Fanuc KAREL source: kc00049.KL

-- PROVISIONAL review KL for V1013-1; original PC SHA256 6f2dececdb086ac4d14ee3edc9f621b24aaa7305749a3dd8db25e0824419496a
-- Incomplete behavior may be omitted. Consult companion uncertainty JSON. Do not deploy.
PROGRAM KC00049
%NOLOCKGROUP
BEGIN
  -- UNRESOLVED_PC offsets 5-35; opcodes 27,22,22,1C,22,27,9D,31
  -- UNRESOLVED_PC offsets 40-44; opcodes 7F
END KC00049
